TYPE ST_PML_Base_In :
STRUCT
	eCommand				: E_PackMLCommand := E_PackMLCommand.None;
	bCommandChangeRequest	: BOOL;
	eMode					: T_PackMLMode := E_PackMLMode.Unknown;
	bModeChangeRequest	: BOOL;
END_STRUCT
END_TYPE

(* stored: Version 1.1.0.1, ProductVersion 3.1.4026.18
   DUT ST_PML_Base_In: Id {4246412d-a49e-46da-bde0-12a192d5b6b4} *)
